FUNCTION_BLOCK AUI2_TO_AUI (* Composite FB for convert bidirectional AUI2 to unidirectional AUI *)
  (* Standard: 61499-2; Function: AUI2_BIDIR forwards its incoming (EO1) side out as a plain unidirectional signal via AUI_OUT. AUI_IN publishes its value onto the outgoing (EI1) side of AUI2_BIDIR.; Description: Copyright (c) 2026 HR Agrartechnik GmbH This program and the accompanying materials are made available under the terms of the Eclipse Public License 2.0 which is available at https://www.eclipse.org/legal/epl-2.0/ SPDX-License-Identifier: EPL-2.0 *)
  (* Version 1.0, 2026-09-12, Franz Höpfinger, HR Agrartechnik GmbH, Initial Version - Konvertierungsfamilie vervollstaendigt (analog zu AR2/AB2/AE2). *)
  PACKAGE adapter::conversion::bidirectional;
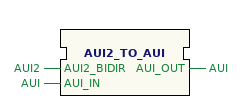
  SOCKETS
    AUI2_BIDIR : adapter::types::bidirectional::AUI2; (* Adapter Input: bidirectional tap, incoming side forwarded to AUI_OUT, outgoing side driven by AUI_IN *)
    AUI_IN : adapter::types::unidirectional::AUI; (* Adapter Input: unidirectional source *)
  END_SOCKETS
  PLUGS
    AUI_OUT : adapter::types::unidirectional::AUI; (* Adapter Output: mirrors AUI2_BIDIR's incoming (indication) side *)
  END_PLUGS
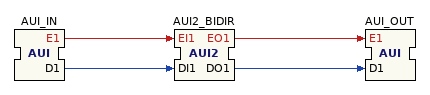
  EVENT_CONNECTIONS
    AUI2_BIDIR.EO1 TO AUI_OUT.E1;
    AUI_IN.E1 TO AUI2_BIDIR.EI1;
  END_CONNECTIONS
  DATA_CONNECTIONS
    AUI2_BIDIR.DO1 TO AUI_OUT.D1;
    AUI_IN.D1 TO AUI2_BIDIR.DI1;
  END_CONNECTIONS
END_FUNCTION_BLOCK
